// TIA Portal V21 export
TYPE "LBC_typeAnalogScaleValues"
TITLE = LBC_typeAnalogScaleValues
// Module related monitoring information
   STRUCT
      enable { ExternalWritable := 'False'} : Bool;   // Enable functionality of FB
      referenceDesignator { ExternalWritable := 'False'} : WString[154];   // Reference Designator for the module incl. its parent
      simulation { ExternalWritable := 'False'} : Bool;   // Enable simulation input of input value
      inputValue { ExternalWritable := 'False'} : LReal;   // Value to be converted
      outputValue { ExternalWritable := 'False'} : LReal;   // Processed and scaled value
      minValueReached { ExternalWritable := 'False'} : Bool;   // Minimum configured process value reached. Value is limited to the minimum configured value.
      maxValueReached { ExternalWritable := 'False'} : Bool;   // Maximum configured process value reached. Value is limited to the maximum configured value.
      error { ExternalWritable := 'False'} : Bool;   // An error occurred while processing the FB
      status { ExternalWritable := 'False'} : Word;   // 16#0000-16#7FFF: Status of the FB 16#8000-16#FFFF: Error identification
   END_STRUCT;
END_TYPE
